(* PLC project Aufgabenserie_3, Beckhoff Automation GmbH TwinCAT PLC Control 3.5.10.30 *)
(* stored: creationDateTime 2018-11-22T20:16:21.5812716, modificationDateTime 2018-11-22T20:16:21.5882738 *)

{attribute 'qualified_only'}
{attribute 'strict'}
TYPE FSM_Deb :
(
	deb_state_init := 0,
	deb_state_low,
	deb_state_rising,
	deb_state_high,
	deb_state_doble_activ,
	deb_state_falling
);
END_TYPE
